(* PLC project Unnamed, Unknown Unnamed 1 *)
(* stored: creationDateTime 2026-05-02T16:14:51, modificationDateTime 2026-05-03T20:15:31 *)

PROGRAM Project_05_Pump_Station_with_PID_Pressure_Control_and_VFD
  VAR
    PB_EStop AT %IX0.0 : BOOL;
    PB_FaultReset AT %IX0.1 : BOOL;
    SW_ModeAuto AT %IX0.2 : BOOL;
    SW_ModeTest AT %IX0.3 : BOOL;
    F2_P1_Overload AT %IX0.4 : BOOL;
    F3_P2_Overload AT %IX0.5 : BOOL;
    KM1_P1_Feedback AT %IX0.6 : BOOL;
    KM2_P2_Feedback AT %IX0.7 : BOOL;
    VFD1_Running AT %IX1.0 : BOOL;
    VFD1_Fault AT %IX1.1 : BOOL;
    LS_SumpLow AT %IX1.2 : BOOL;
    PB_P1_ManStart AT %IX1.3 : BOOL;
    PB_P1_ManStop AT %IX1.4 : BOOL;
    PB_P2_ManStart AT %IX1.5 : BOOL;
    PB_P2_ManStop AT %IX1.6 : BOOL;
    LS_TankHighHigh AT %IX1.7 : BOOL;
    KM1_P1_Contactor AT %QX0.0 : BOOL;
    KM2_P2_Contactor AT %QX0.1 : BOOL;
    VFD1_Enable AT %QX0.2 : BOOL;
    SOL_DischargeValve AT %QX0.3 : BOOL;
    HL1_P1RunLamp AT %QX0.4 : BOOL;
    HL2_P2RunLamp AT %QX0.5 : BOOL;
    HL3_AlarmLamp AT %QX0.6 : BOOL;
    HL4_AutoLamp AT %QX0.7 : BOOL;
    BZ1_Alarm AT %QX1.0 : BOOL;
    AI_Pressure_Raw AT %IW0 : INT;
    AI_Flow_Raw AT %IW1 : INT;
    AI_VFD1_Speed_Raw AT %IW2 : INT;
    AO_VFD1_SpeedRef AT %QW0 : INT;
  END_VAR
  VAR
    MasterEnable : BOOL;
    FaultActive : BOOL;
    FaultP1_Overload : BOOL;
    FaultP2_Overload : BOOL;
    FaultVFD1 : BOOL;
    FaultSumpLow : BOOL;
    FaultPressLow : BOOL;
    FaultPressHigh : BOOL;
    AutoMode : BOOL;
    ManualMode : BOOL;
    TestMode : BOOL;
    P1_RunCmd : BOOL;
    P2_RunCmd : BOOL;
    P2_LagActive : BOOL;
    DutySwapReq : BOOL;
    BuzzerSilenced : BOOL;
    Clock_1Hz : BOOL;
    Pressure_EU : REAL;
    Flow_EU : REAL;
    VFD1_Speed_EU : REAL;
    Setpoint_EU : REAL := = 6.0;
    PID_Output : REAL := = 20.0;
    ManSpeedRef : REAL := = 50.0;
    P2_LagThreshold : REAL := = 95.0;
    P2_StopThreshold : REAL := = 60.0;
    PressAlarmLo : REAL := = 4.0;
    PressAlarmHi : REAL := = 12.0;
    Pressure_Raw_Real : REAL;
    Pressure_Mul : REAL;
    Flow_Raw_Real : REAL;
    Flow_Mul : REAL;
    VFD_Raw_Real : REAL;
    VFD_Mul : REAL;
    PressAlarmLo_Reset : REAL := = 4.3;
    PressAlarmHi_Reset : REAL := = 11.5;
    AO_TempReal : REAL;
    AO_TempReal2 : REAL;
    P2_StartPressure : REAL;
    P2_SpeedHigh : BOOL;
    P2_PressureLow : BOOL;
    P2_SpeedLow : BOOL;
    RuntimeDiff : REAL;
    FlowPerSecond : REAL;
    FaultP1_Feedback : BOOL;
    FaultP2_Feedback : BOOL;
    P1_RunHours : REAL := = 0.0;
    P2_RunHours : REAL := = 0.0;
    FlowTotal_Daily : REAL := = 0.0;
    P1_StartCount : INT := = 0.0;
    P2_StartCount : INT := = 0.0;
    I6 : REAL := = 16;
    n27648 : REAL := = 27648.0;
    TON_PressAlarmDelay : TON;
    TON_PressAlarmDelayTime : TIME := T#10s;
    TON_P2_StartDelayTime : TIME := T#5s;
    n200 : REAL := = 200.0;
    n100 : REAL := = 100.0;
    nClock : REAL := = 0.000278;
    n20 : REAL := = 20.0;
    n10 : REAL := = 10.0;
    n0 : REAL := = 0;
    n05 : REAL := = 0.5;
    n3600 : REAL := = 3600.0;
    TON_ValvePreOpen : TON;
    TON_ValvePreOpenTime : TIME := = T#3s;
    TON_P1_FbkDelayTime : TIME := = T#1s;
    TON_P2_StopDelayTime : TIME := =T#30s;
    TON_P2_FbkDelayTime : TIME := =T#1s;
    TON_P1_FbkDelay : TON;
    PID0 : PID;
    PID_TR : REAL := = 30.0;
    PID_TD : REAL := = 0.0;
    PID_CYCLE : REAL;
    PID_LowLimit : REAL;
    PID_HighLimit : REAL;
    TON_P2_StartDelay : TON;
    TON_P2_StopDelay : TON;
    TON_P2_FbkDelay : TON;
  END_VAR

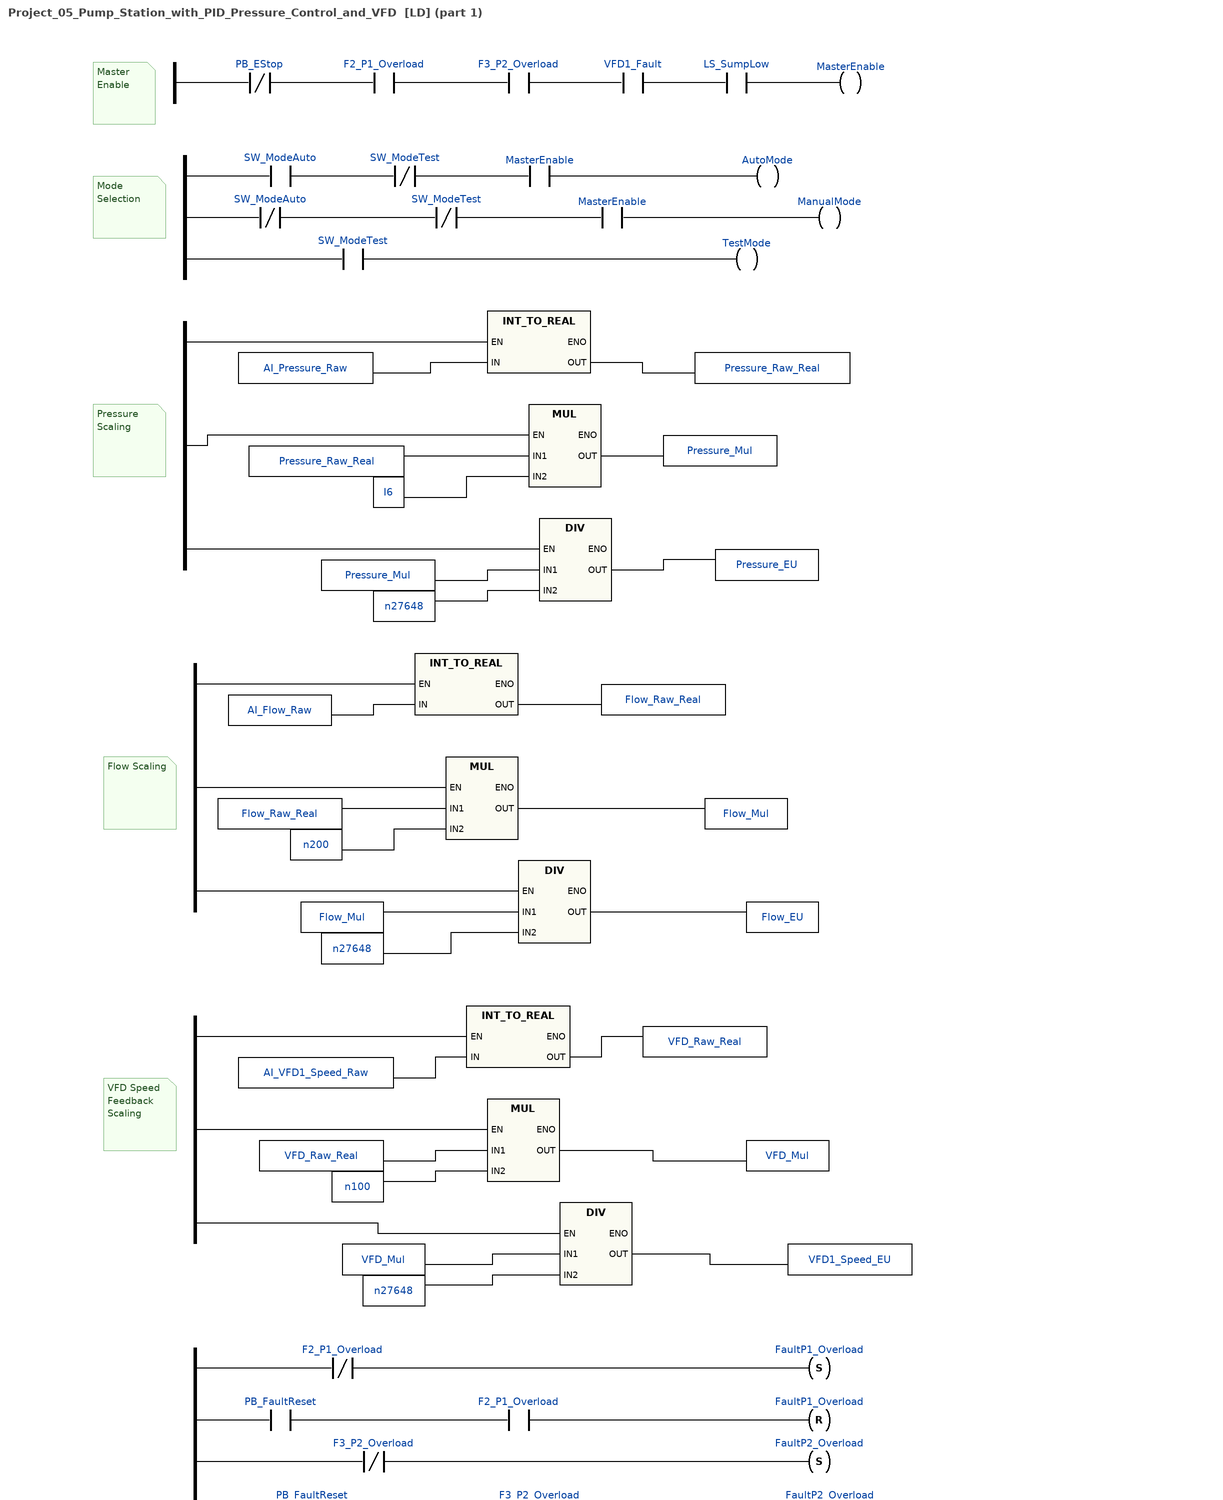
(* LD diagram, written out as Structured Text *)
(* Master Enable *)
MasterEnable := NOT PB_EStop AND F2_P1_Overload AND F3_P2_Overload AND VFD1_Fault AND LS_SumpLow;
AutoMode := SW_ModeAuto AND NOT SW_ModeTest AND MasterEnable;
(* Mode Selection *)
ManualMode := NOT SW_ModeAuto AND NOT SW_ModeTest AND MasterEnable;
TestMode := SW_ModeTest;
(* Pressure Scaling *)
(* Flow Scaling *)
(* VFD Speed Feedback Scaling *)
IF NOT F2_P1_Overload THEN FaultP1_Overload := TRUE; END_IF;
IF PB_FaultReset AND F2_P1_Overload THEN FaultP1_Overload := FALSE; END_IF;
IF NOT F3_P2_Overload THEN FaultP2_Overload := TRUE; END_IF;
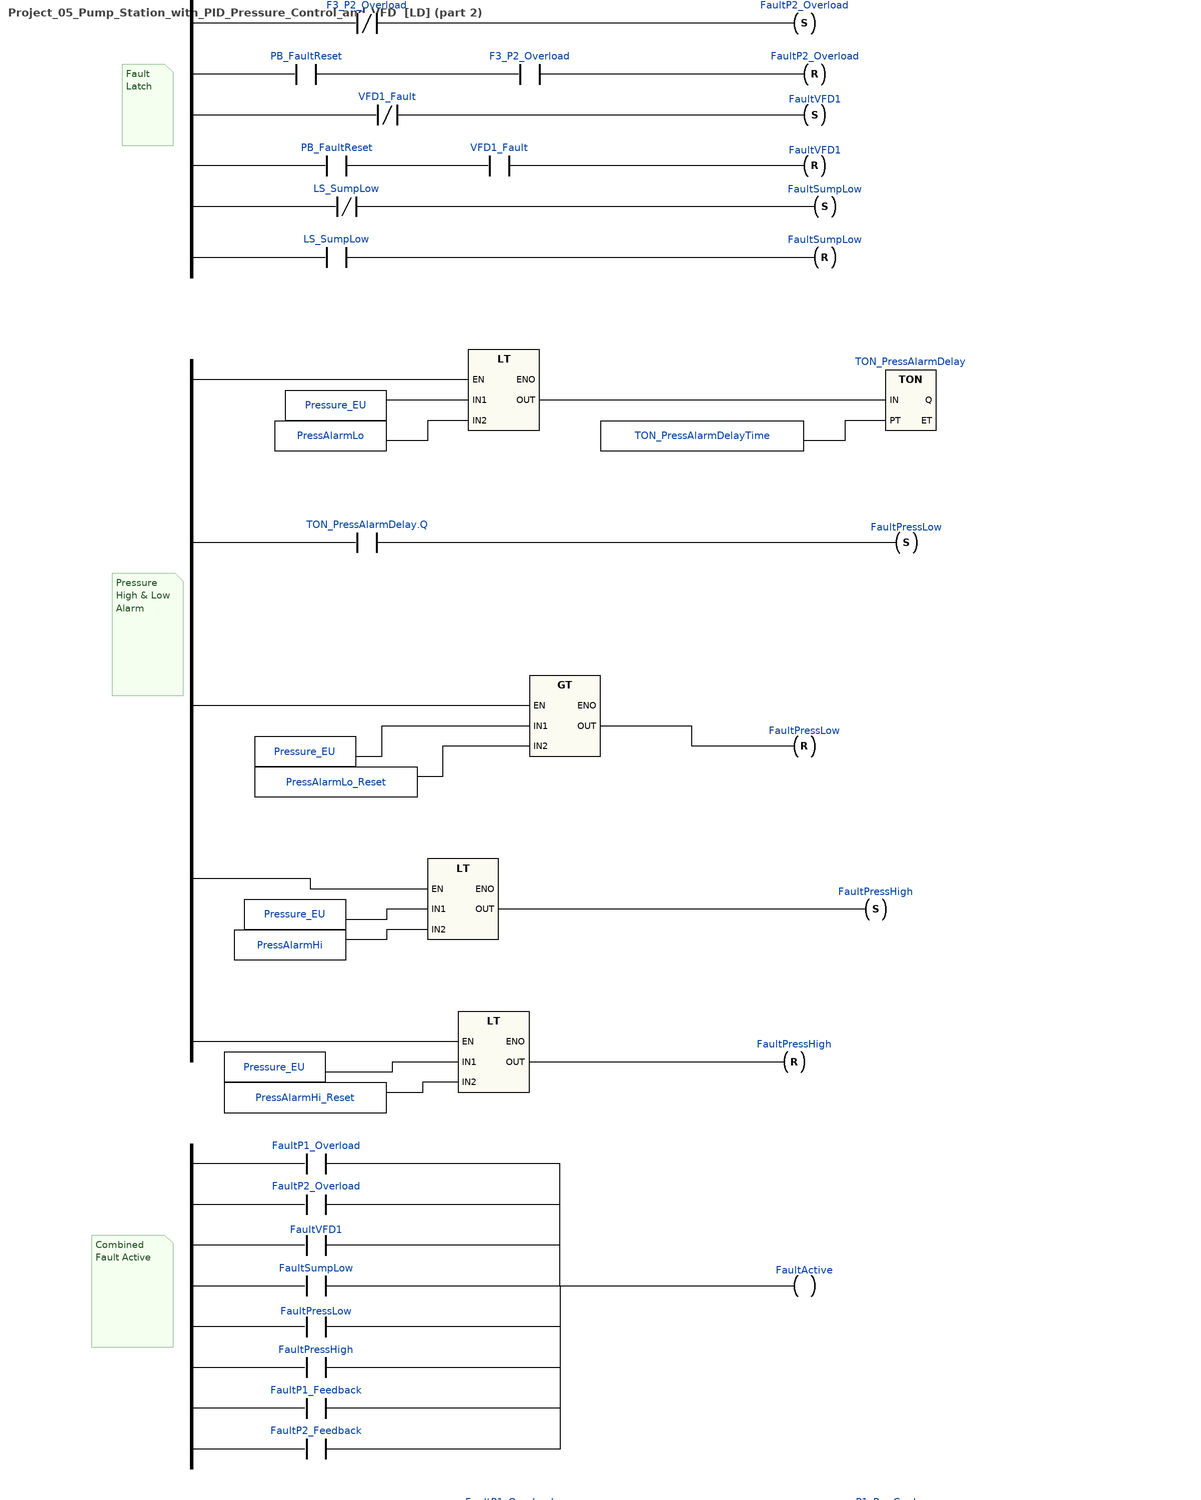
(* Fault Latch *)
IF PB_FaultReset AND F3_P2_Overload THEN FaultP2_Overload := FALSE; END_IF;
IF NOT VFD1_Fault THEN FaultVFD1 := TRUE; END_IF;
IF PB_FaultReset AND VFD1_Fault THEN FaultVFD1 := FALSE; END_IF;
IF NOT LS_SumpLow THEN FaultSumpLow := TRUE; END_IF;
IF LS_SumpLow THEN FaultSumpLow := FALSE; END_IF;
Pressure_Raw_Real := INT_TO_REAL(AI_Pressure_Raw);
Pressure_Mul := Pressure_Raw_Real * I6;
Pressure_EU := Pressure_Mul / n27648;
IF TON_PressAlarmDelay.Q THEN FaultPressLow := TRUE; END_IF;
Flow_Raw_Real := INT_TO_REAL(AI_Flow_Raw);
Flow_Mul := Flow_Raw_Real * n200;
Flow_EU := Flow_Mul / n27648;
VFD_Raw_Real := INT_TO_REAL(AI_VFD1_Speed_Raw);
VFD_Mul := VFD_Raw_Real * n100;
VFD1_Speed_EU := VFD_Mul / n27648;
(* Pressure High & Low Alarm *)
IF Pressure_EU > PressAlarmLo_Reset THEN FaultPressLow := FALSE; END_IF;
IF Pressure_EU < PressAlarmHi THEN FaultPressHigh := TRUE; END_IF;
IF Pressure_EU < PressAlarmHi_Reset THEN FaultPressHigh := FALSE; END_IF;
(* Combined Fault Active *)
FaultActive := FaultSumpLow OR FaultP1_Overload OR FaultP2_Overload OR FaultVFD1 OR FaultPressLow OR FaultPressHigh OR FaultP1_Feedback OR FaultP2_Feedback;
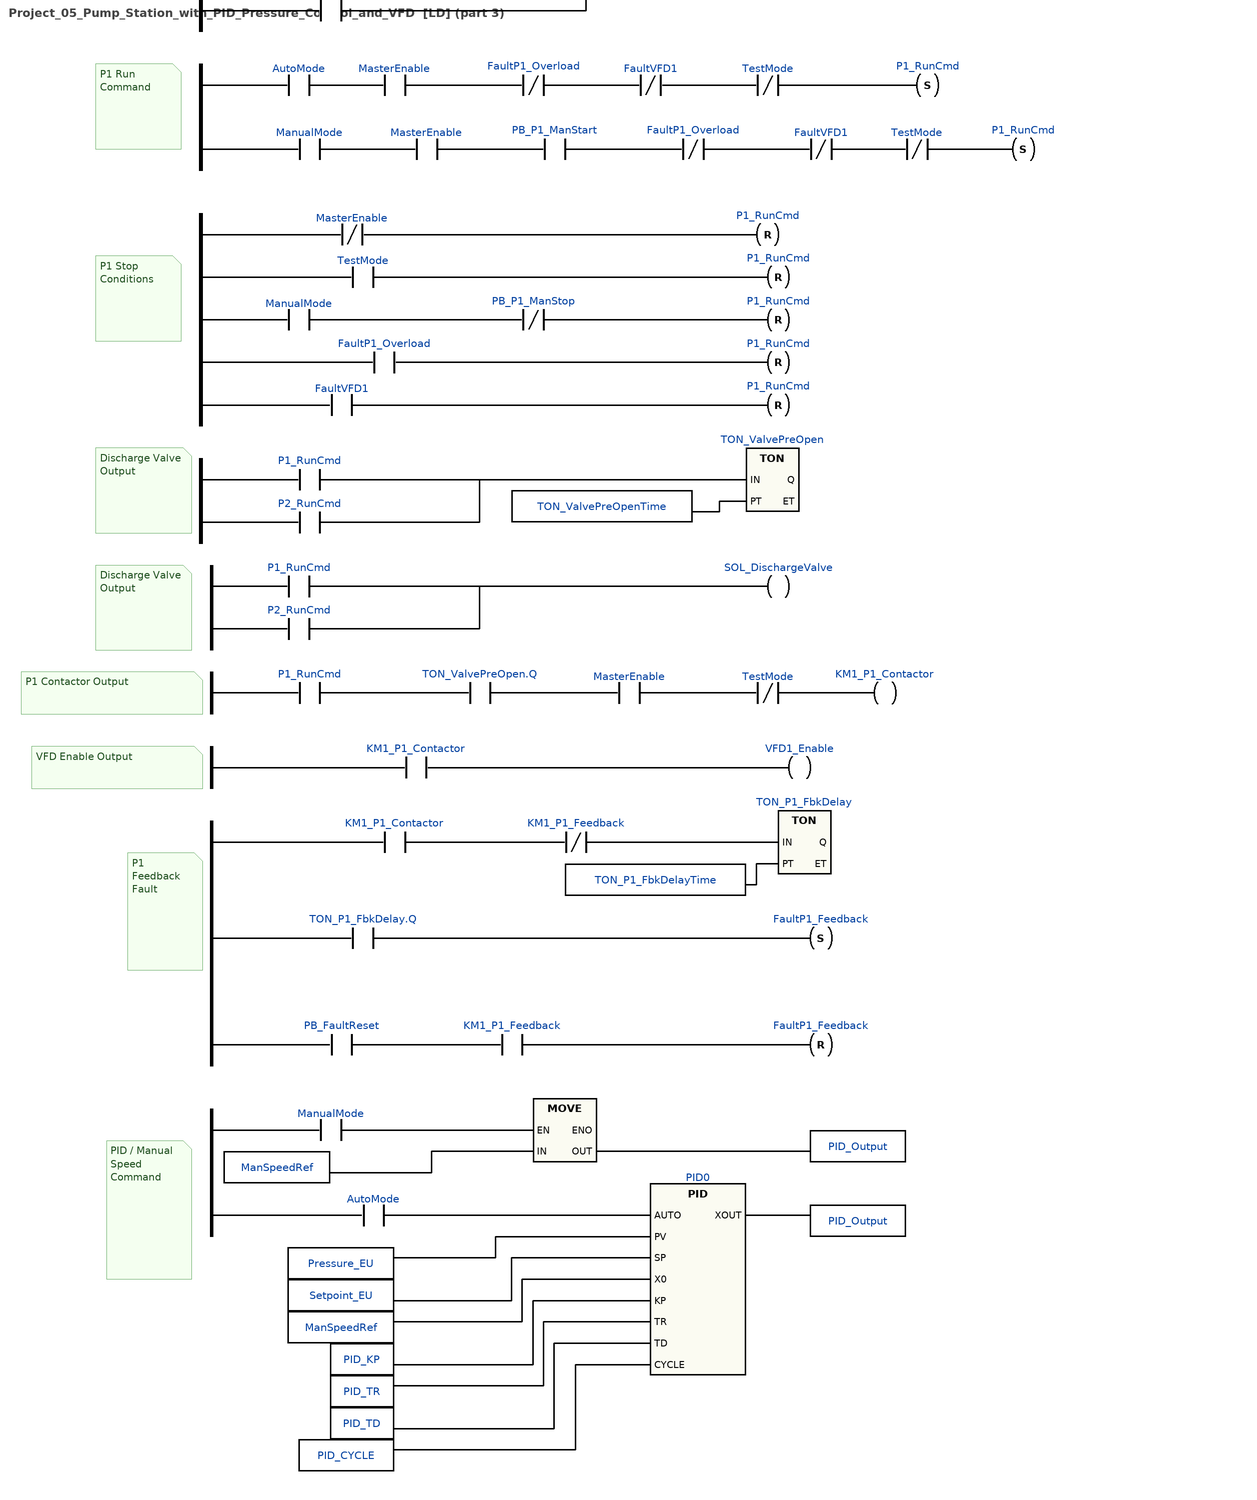
(* P1 Run Command *)
IF AutoMode AND MasterEnable AND NOT FaultP1_Overload AND NOT FaultVFD1 AND NOT TestMode THEN P1_RunCmd := TRUE; END_IF;
IF ManualMode AND MasterEnable AND PB_P1_ManStart AND NOT FaultP1_Overload AND NOT FaultVFD1 AND NOT TestMode THEN P1_RunCmd := TRUE; END_IF;
(* P1 Stop Conditions *)
IF TestMode THEN P1_RunCmd := FALSE; END_IF;
IF NOT MasterEnable THEN P1_RunCmd := FALSE; END_IF;
IF ManualMode AND NOT PB_P1_ManStop THEN P1_RunCmd := FALSE; END_IF;
IF FaultP1_Overload THEN P1_RunCmd := FALSE; END_IF;
IF FaultVFD1 THEN P1_RunCmd := FALSE; END_IF;
(* Discharge Valve Output *)
(* Discharge Valve Output *)
SOL_DischargeValve := P1_RunCmd OR P2_RunCmd;
(* P1 Contactor Output *)
KM1_P1_Contactor := P1_RunCmd AND TON_ValvePreOpen.Q AND MasterEnable AND NOT TestMode;
(* VFD Enable Output *)
VFD1_Enable := KM1_P1_Contactor;
(* P1 Feedback Fault *)
IF TON_P1_FbkDelay.Q THEN FaultP1_Feedback := TRUE; END_IF;
IF PB_FaultReset AND KM1_P1_Feedback THEN FaultP1_Feedback := FALSE; END_IF;
IF ManualMode THEN PID_Output := ManSpeedRef; END_IF;
(* PID / Manual Speed Command *)
PID0(AUTO := AutoMode, PV := Pressure_EU, SP := Setpoint_EU, X0 := ManSpeedRef, KP := PID_KP, TR := PID_TR, TD := PID_TD, CYCLE := PID_CYCLE);
PID_Output := PID0.XOUT;
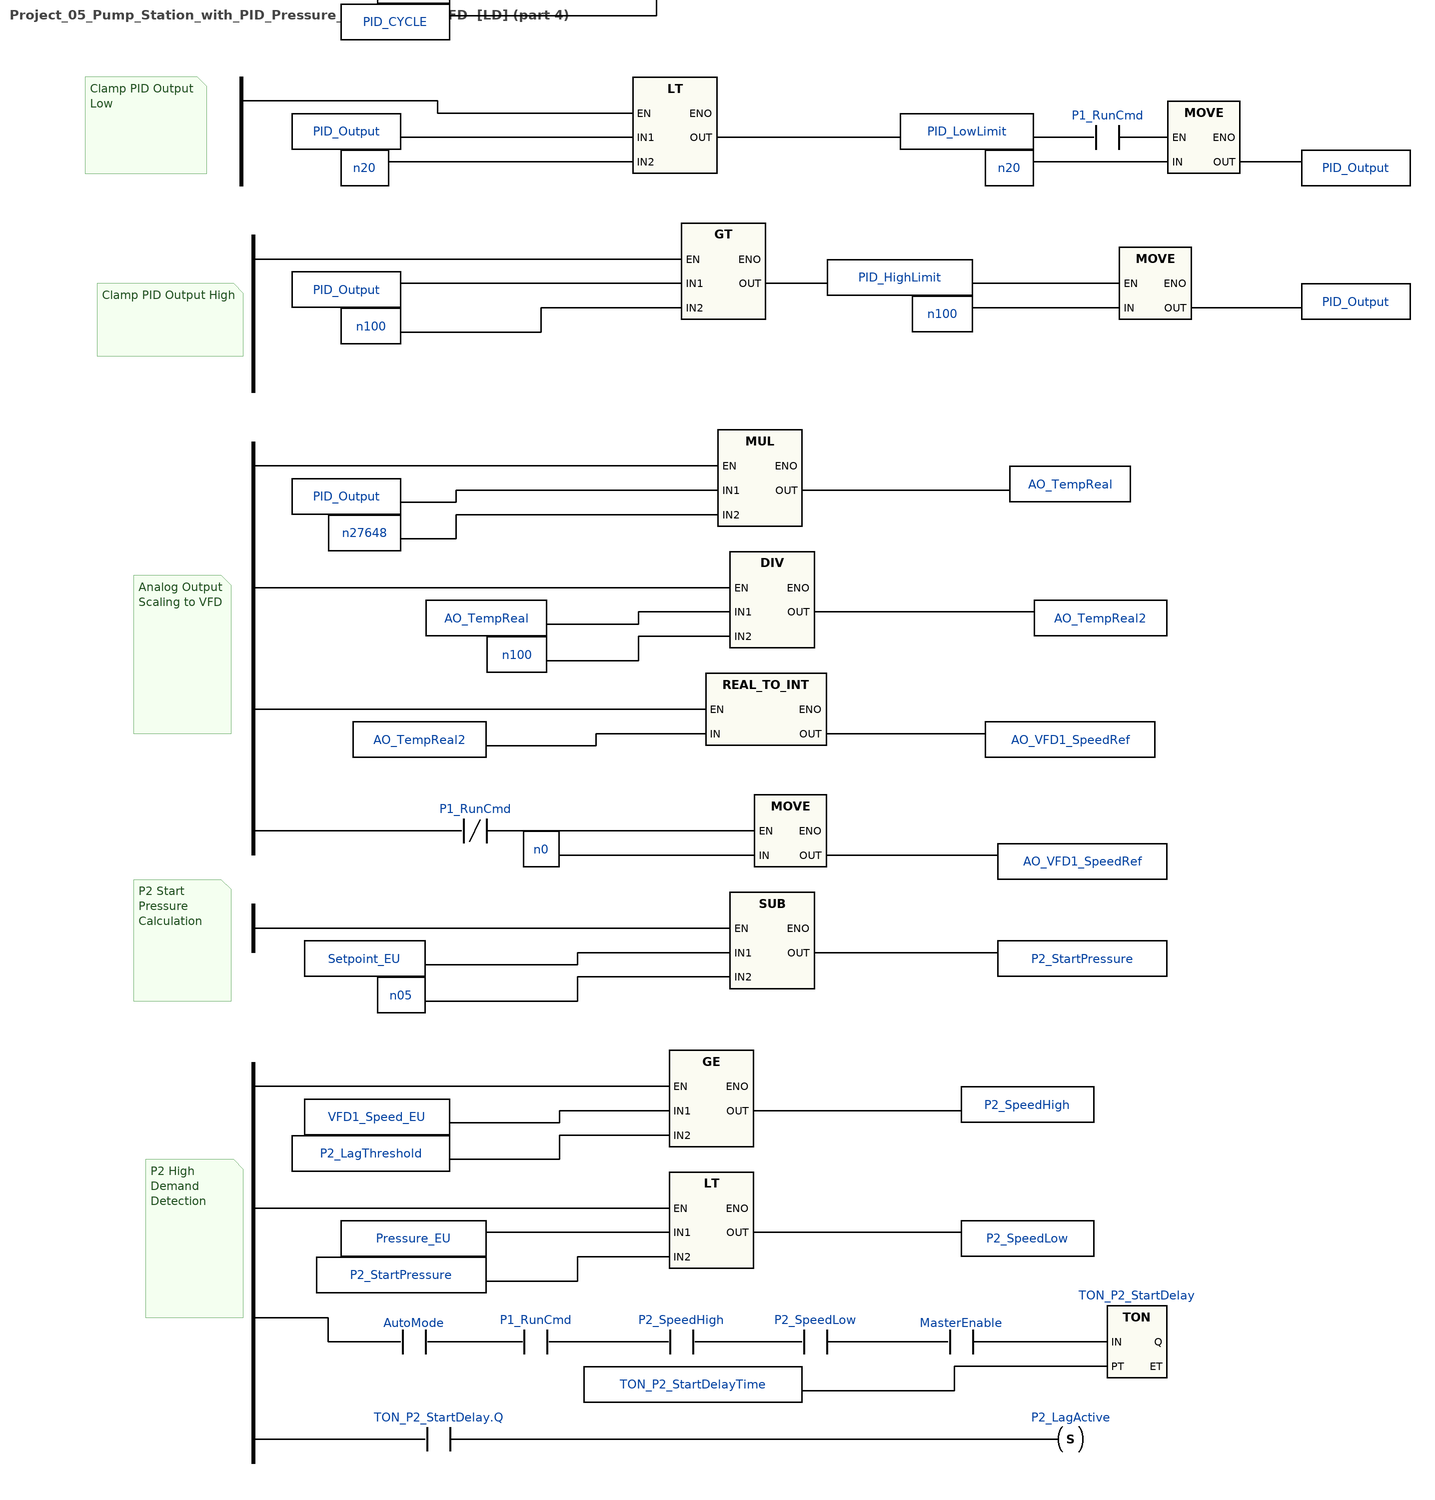
(* Clamp PID Output Low *)
PID_LowLimit := PID_Output < n20;
IF PID_LowLimit AND P1_RunCmd THEN PID_Output := n20; END_IF;
PID_HighLimit := PID_Output > n100;
(* Clamp PID Output High *)
IF PID_HighLimit THEN PID_Output := n100; END_IF;
AO_TempReal := PID_Output * n27648;
(* Analog Output Scaling to VFD *)
AO_TempReal2 := AO_TempReal / n100;
AO_VFD1_SpeedRef := REAL_TO_INT(AO_TempReal2);
IF NOT P1_RunCmd THEN AO_VFD1_SpeedRef := n0; END_IF;
(* P2 Start Pressure Calculation *)
P2_StartPressure := Setpoint_EU - n05;
P2_SpeedHigh := VFD1_Speed_EU >= P2_LagThreshold;
(* P2 High Demand Detection *)
P2_SpeedLow := Pressure_EU < P2_StartPressure;
IF TON_P2_StartDelay.Q THEN P2_LagActive := TRUE; END_IF;
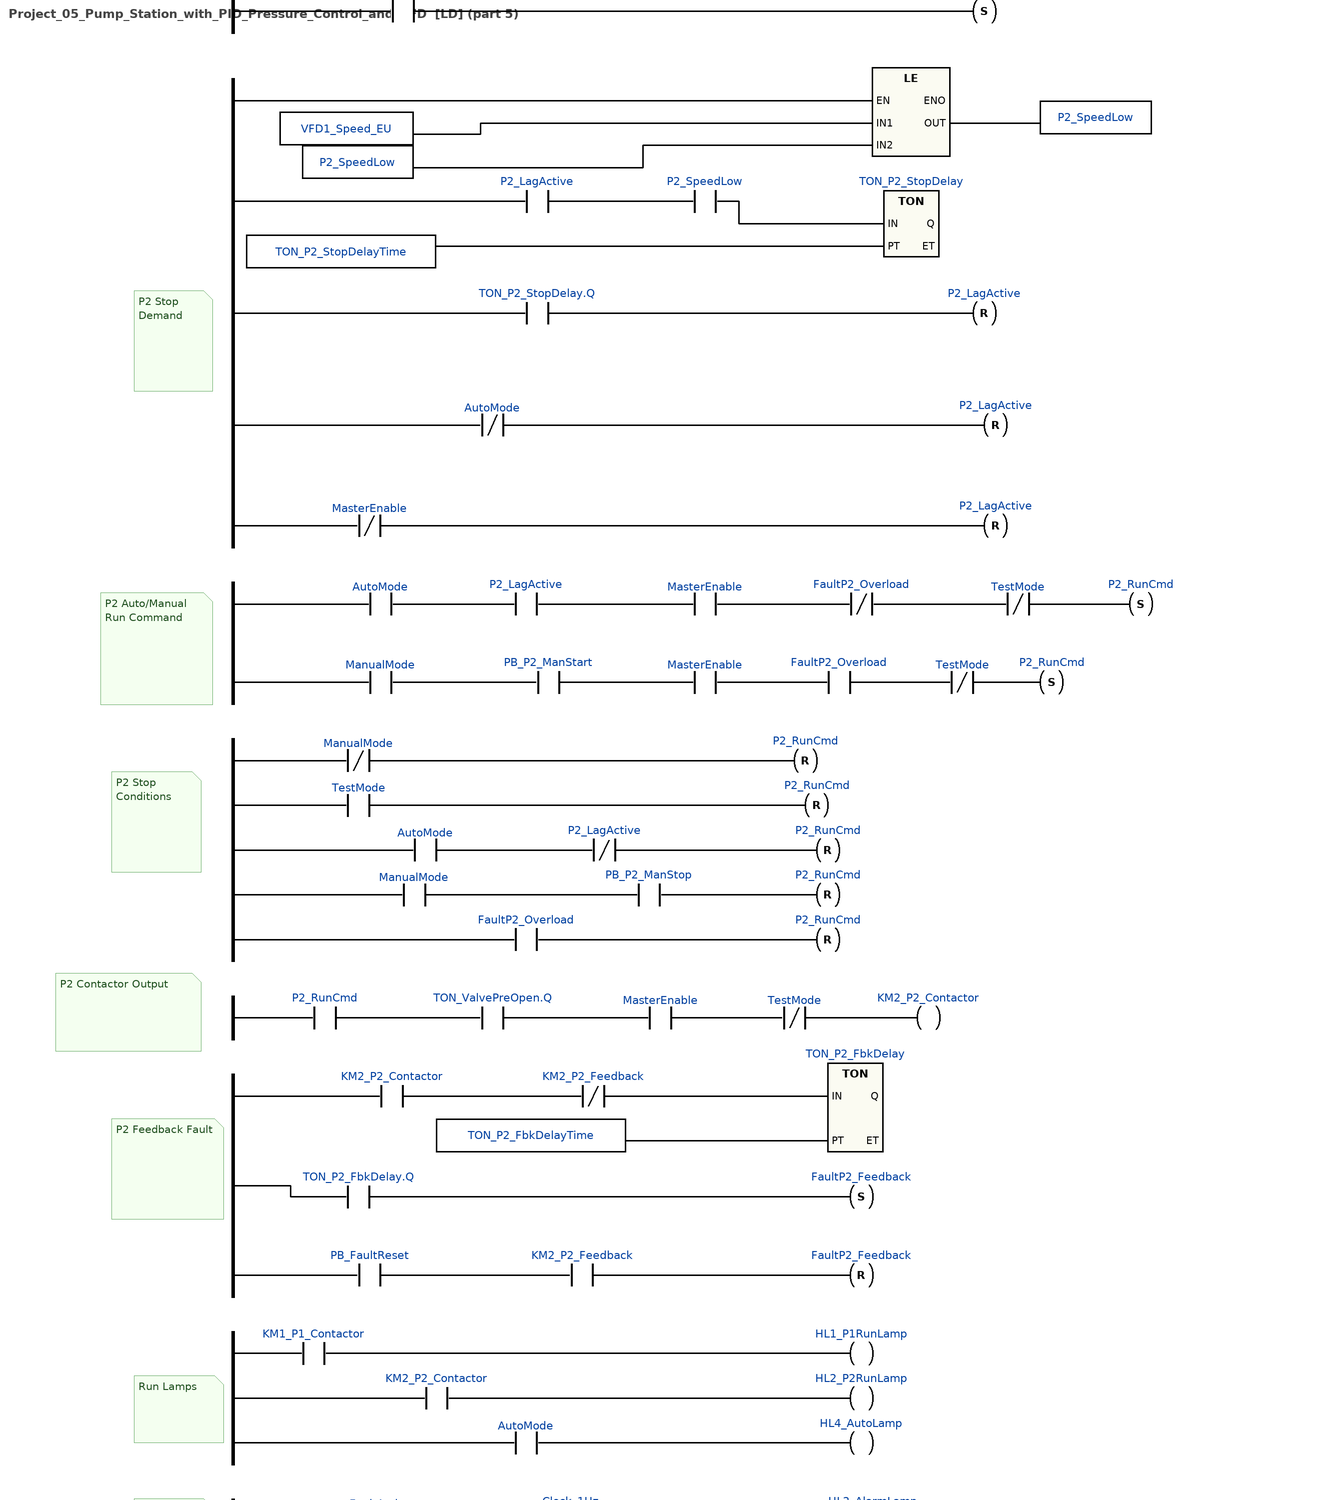
P2_SpeedLow := VFD1_Speed_EU <= P2_SpeedLow;
(* P2 Stop Demand *)
IF TON_P2_StopDelay.Q THEN P2_LagActive := FALSE; END_IF;
IF NOT AutoMode THEN P2_LagActive := FALSE; END_IF;
IF NOT MasterEnable THEN P2_LagActive := FALSE; END_IF;
(* P2 Auto/Manual Run Command *)
IF AutoMode AND P2_LagActive AND MasterEnable AND NOT FaultP2_Overload AND NOT TestMode THEN P2_RunCmd := TRUE; END_IF;
IF ManualMode AND PB_P2_ManStart AND MasterEnable AND FaultP2_Overload AND NOT TestMode THEN P2_RunCmd := TRUE; END_IF;
(* P2 Stop Conditions *)
IF TestMode THEN P2_RunCmd := FALSE; END_IF;
IF NOT ManualMode THEN P2_RunCmd := FALSE; END_IF;
IF AutoMode AND NOT P2_LagActive THEN P2_RunCmd := FALSE; END_IF;
IF ManualMode AND PB_P2_ManStop THEN P2_RunCmd := FALSE; END_IF;
IF FaultP2_Overload THEN P2_RunCmd := FALSE; END_IF;
(* P2 Contactor Output *)
KM2_P2_Contactor := P2_RunCmd AND TON_ValvePreOpen.Q AND MasterEnable AND NOT TestMode;
(* P2 Feedback Fault *)
IF TON_P2_FbkDelay.Q THEN FaultP2_Feedback := TRUE; END_IF;
IF PB_FaultReset AND KM2_P2_Feedback THEN FaultP2_Feedback := FALSE; END_IF;
HL1_P1RunLamp := KM1_P1_Contactor;
(* Run Lamps *)
HL2_P2RunLamp := KM2_P2_Contactor;
HL4_AutoLamp := AutoMode;
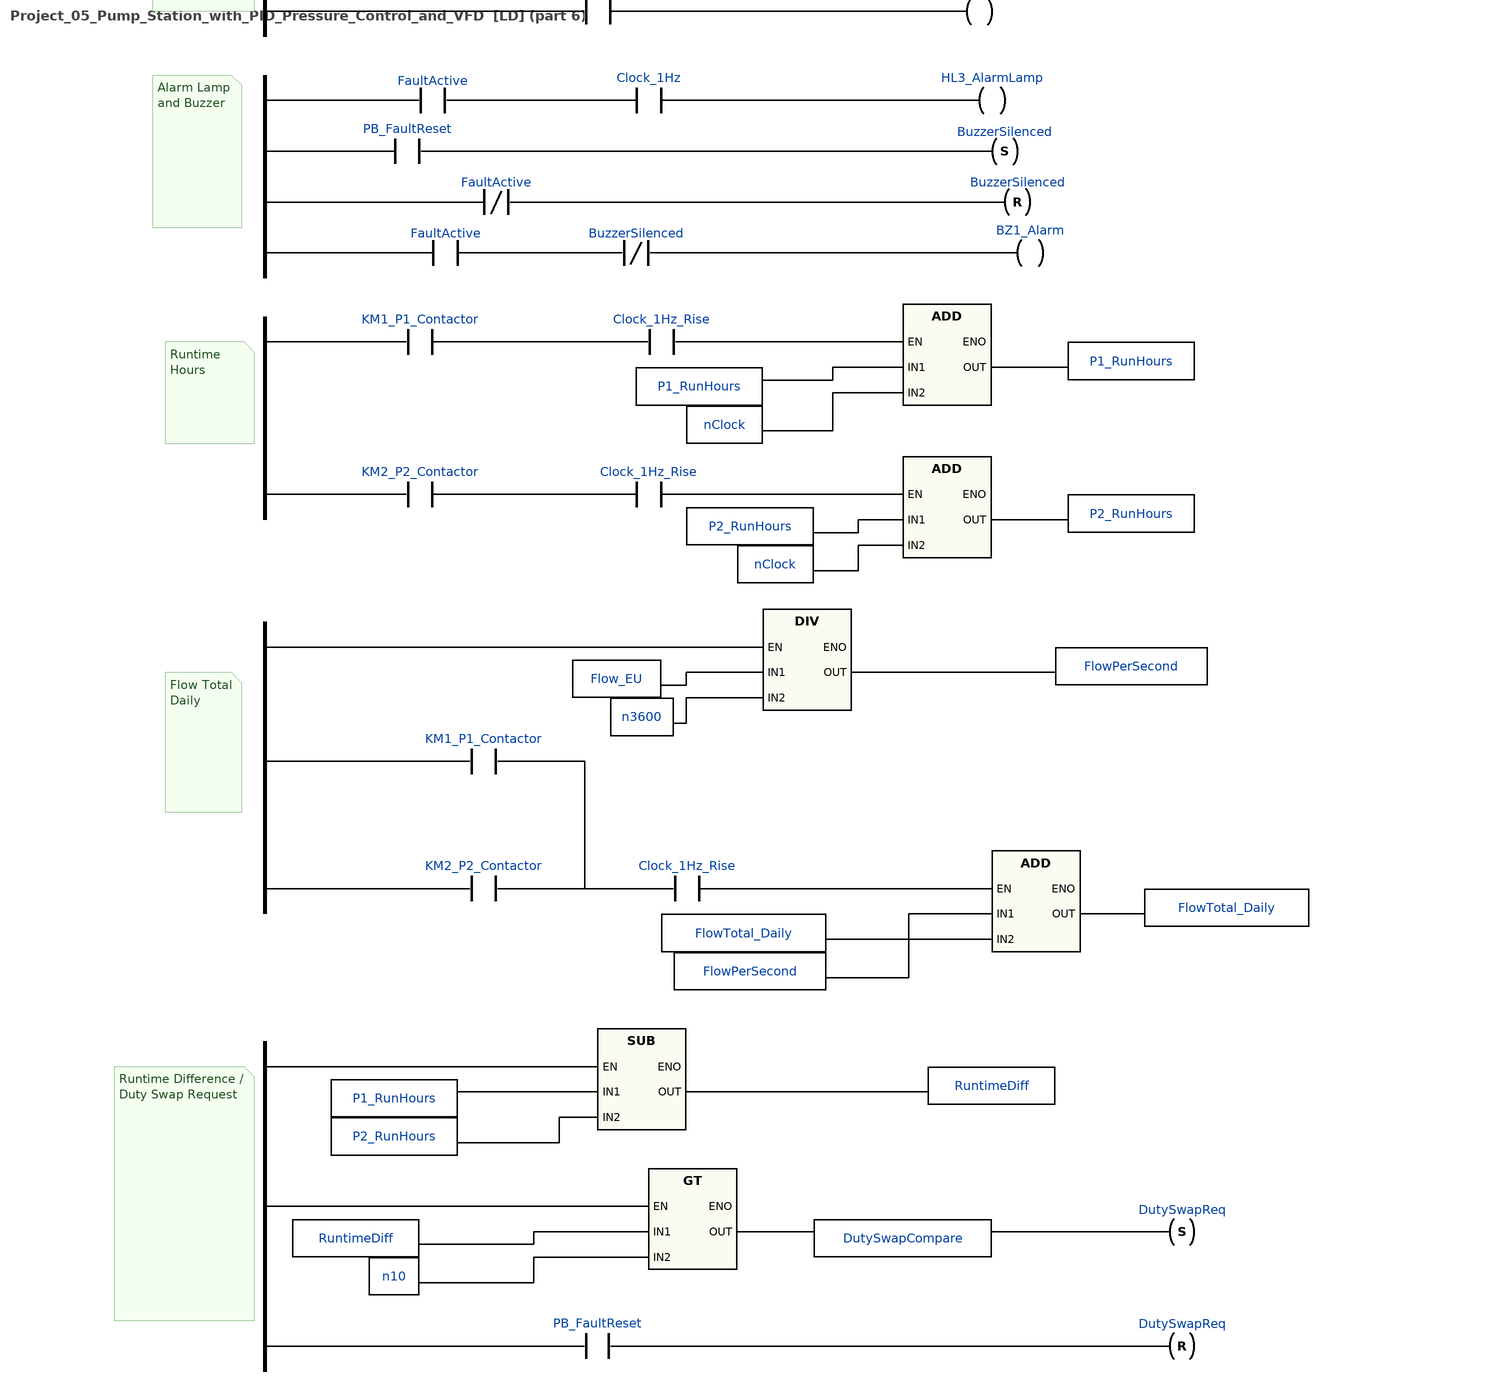
(* Alarm Lamp and Buzzer *)
HL3_AlarmLamp := FaultActive AND Clock_1Hz;
IF PB_FaultReset THEN BuzzerSilenced := TRUE; END_IF;
IF NOT FaultActive THEN BuzzerSilenced := FALSE; END_IF;
BZ1_Alarm := FaultActive AND NOT BuzzerSilenced;
(* Runtime Hours *)
IF KM1_P1_Contactor AND Clock_1Hz_Rise THEN P1_RunHours := P1_RunHours + nClock; END_IF;
IF KM2_P2_Contactor AND Clock_1Hz_Rise THEN P2_RunHours := P2_RunHours + nClock; END_IF;
FlowPerSecond := Flow_EU / n3600;
(* Flow Total Daily *)
IF (KM2_P2_Contactor OR KM1_P1_Contactor) AND Clock_1Hz_Rise THEN FlowTotal_Daily := FlowTotal_Daily + FlowPerSecond; END_IF;
(* Runtime Difference / Duty Swap Request *)
RuntimeDiff := P1_RunHours - P2_RunHours;
DutySwapCompare := RuntimeDiff > n10;
IF DutySwapCompare THEN DutySwapReq := TRUE; END_IF;
IF PB_FaultReset THEN DutySwapReq := FALSE; END_IF;
TON_PressAlarmDelay(IN := Pressure_EU < PressAlarmLo, PT := TON_PressAlarmDelayTime);
TON_ValvePreOpen(IN := P1_RunCmd OR P2_RunCmd, PT := TON_ValvePreOpenTime);
TON_P1_FbkDelay(IN := KM1_P1_Contactor AND NOT KM1_P1_Feedback, PT := TON_P1_FbkDelayTime);
TON_P2_StartDelay(IN := AutoMode AND P1_RunCmd AND P2_SpeedHigh AND P2_SpeedLow AND MasterEnable, PT := TON_P2_StartDelayTime);
TON_P2_StopDelay(IN := P2_LagActive AND P2_SpeedLow, PT := TON_P2_StopDelayTime);
TON_P2_FbkDelay(IN := KM2_P2_Contactor AND NOT KM2_P2_Feedback, PT := TON_P2_FbkDelayTime);
END_PROGRAM

CONFIGURATION Config0
  RESOURCE Res0 ON PLC
    TASK task0(INTERVAL := T#20ms, PRIORITY := 0);
    PROGRAM instance0 WITH task0 : Project_05_Pump_Station_with_PID_Pressure_Control_and_VFD;
  END_RESOURCE
END_CONFIGURATION
